Staubli VAL3: NoCloseShape.pgx

public program NoCloseShape(point& x_pCut[], point& x_pMC[], bool& x_bMC[], num x_nLength, bool& x_bRes)
  local num l_nNum
  local trsf l_trBuff[3]
  local trsf l_trTe
  local num l_nArc
  local num l_nLength
begin
  //获得切割的真正长度是多少



  x_bRes=false
  //  x_nLength=0
  if size(x_pCut)!=size(x_pMC) or size(x_pCut)!=size(x_bMC)
    return
  endIf

  //如果只有一个点，则退出
  if size(x_bMC)==1
    //  x_bRes=true
    return
  endIf


  //多于一个点进行计算
  l_nNum=size(x_bMC)-1
  if !x_bMC[l_nNum]
    l_nLength=distance(x_pCut[l_nNum-1].trsf,x_pCut[l_nNum].trsf)

  else
    l_trBuff[0]=x_pCut[l_nNum-1].trsf
    l_trBuff[1]=x_pMC[l_nNum].trsf
    l_trBuff[2]=x_pCut[l_nNum].trsf
    //获取圆弧长度
    call GetArcLength(l_trBuff,l_nLength,x_bRes)
    if !x_bRes
      return
    endIf

  endIf

  if x_nLength>l_nLength
    x_bRes=false
    return
  endIf

  if !x_bMC[l_nNum]
    l_trTe=interpolateL(x_pCut[l_nNum-1].trsf,x_pCut[l_nNum].trsf,x_nLength/l_nLength)
    x_pCut[l_nNum].trsf=l_trTe
  else

    l_trTe=interpolateC(x_pCut[l_nNum-1].trsf,x_pMC[l_nNum].trsf,x_pCut[l_nNum].trsf,x_nLength/l_nLength)
    //保证其是小于180度的圆弧
    if distance(l_trTe,x_pCut[l_nNum-1].trsf)<=distance(x_pMC[l_nNum].trsf,x_pCut[l_nNum-1].trsf)
      x_pCut[l_nNum].trsf=x_pMC[l_nNum].trsf
      x_pMC[l_nNum].trsf=l_trTe
    else
      x_pCut[l_nNum].trsf=l_trTe
    endIf



  endIf



  x_bRes=true

end
